Universal Robots PolyScope program: sand2.urp

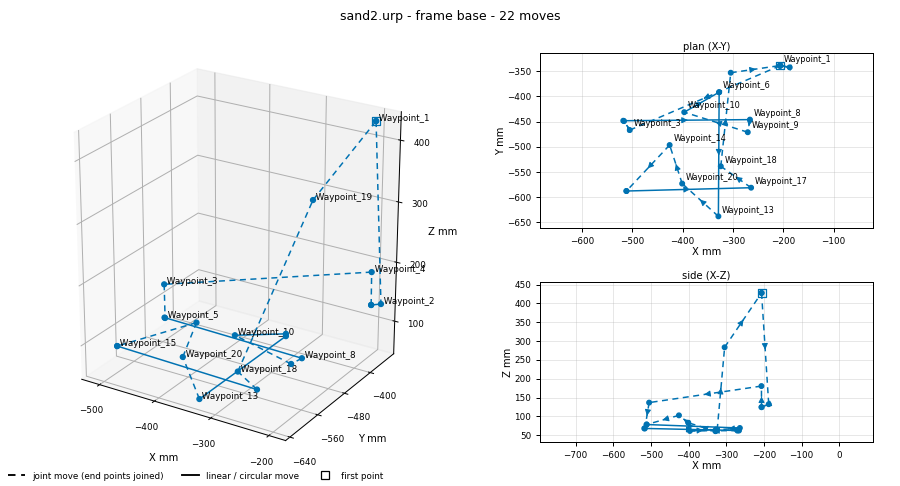
[picture p0: tool path of sand2.urp in frame base, 22 of 22 moves have a stored position in this frame; points joined in program order, loops and branches not executed]
Program sand2 (installation=default directory=/programs/archive createdIn=5.11.5.1010327 lastSavedIn=5.11.5.1010327 robotSerialNumber=20215500677)
Calibrated DH parameters: a=[0.000204, -0.239222, -0.391845, -0.000001, 0.000022, 0]; d=[0.162722, -355.808559, 353.37206, 2.570385, 0.099741, 0.099629]; alpha=[1.571124, 0.000988, 0.008295, 1.568963, -1.570303, 0]; deltaTheta=[0, -0.973091, 7.204745, 0.05153, 0, 0]
Robot Program (runOnlyOnce=false)
  MoveJ speed 60 deg/s, acceleration 80 deg/s^2 (useActiveTCP=true) feature=Base
    Waypoint Waypoint_1: TCP in base x=-206.269 y=-338.618 z=428.007 mm, rx=-2.8182 ry=-1.388 rz=0 rad; joints [-101.561, -74.063, -112.511, -83.459, 90.481, 115.929] deg
    Popup Message (haltProgram=false message=Load the cube inputType=Text)
    Waypoint Waypoint_2: TCP in base x=-187.281 y=-342.265 z=132.578 mm, rx=-2.8182 ry=-1.3882 rz=-0.0001 rad; joints [-98.674, -101.388, -141.016, -27.626, 90.232, 119.185] deg
  MoveL speed 100 mm/s, acceleration 600 mm/s^2 (useActiveTCP=true) feature=Base
    Waypoint Waypoint_7: TCP in base x=-206.272 y=-338.621 z=124.68 mm, rx=-2.8183 ry=-1.388 rz=0 rad; joints [-101.67, -103.53, -140.312, -26.186, 90.22, 116.201] deg
    URCap Finishing Tool Control (Robotiq_Copilot, Robotiq Inc.) dataModel(ToolOutputNameKey=digital_out[0], HackTriggeringContributionIsDefinedMethodKey=true)
    URCap Zero FT Sensor (Robotiq_Copilot, Robotiq Inc.) dataModel(NodeInitializedKey=true, WaitForSteadyWrenchOptionKey=false)
    URCap Find Surface (Robotiq_Copilot, Robotiq Inc.) dataModel(NodeInitializedKey=true, ZeroSensorBeforeKey=true, ls_force=10.0, ls_distance=100.0, ls_speed=5.0, ls_if_distance=false, ls_if_force=false, WaitForSteadyWrenchOptionKey=true); state(isChildrenLocked=true)
      'Add Stop conditions from the Find Surface node'
    Force Simple feature=Joint_6_name; selection=[0, 0, 1, 0, 0, 0]; wrench=[0, 0, 3, 0, 0, 0]; limitsForce=[0.15, 0.15, 0.15, 1.047198, 1.047198, 1.047198]; limitsMotion=[0.1, 0.1, 0.1, 0.349066, 0.349066, 0.349066]
      URCap Path Generator (Robotiq_Copilot, Robotiq Inc.) dataModel(pathOptionsTypeKey=TOOL_ON_ROBOT, coverageModeKey=PERIMETER_ONLY, relativePathKey=true, selectedFeatureNameKey=Actual pose, offsetTypeKey=Actual pose, PathTypeKey=FOUR_POINTS_VERTICAL, WaypointPoseKey1=[-0.20629660419563384, -0.3386300161325113, 0.12467794719703908, -2.8183538684059672, -1.3879313624712748, 7.933958590910351E-5], WaypointJointPositionsKey1=[-1.774516623062409, -1.8069839115661104, -2.4488972349192424, -0.45702049851803395, 1.5746060018745398, 2.028078014086811], WaypointPoseKey3=[-0.21004244357085544, -0.6855155317004626, 0.11340652779835002, 2.8181701273709097, 1.3883207082344338, -1.963602976327567E-4], WaypointJointPositionsKey3=[-1.6808014341985542, -2.3592393235059745, -1.4739016889725134, -0.8796152951918419, 1.5775116439677972, 2.1200337468062562], WaypointPoseKey4=[-0.5667053703425011, -0.6982977977050183, 0.1203185558229202, 2.818031624647423, 1.3883496686721377, -2.3680285315842763E-4], WaypointJointPositionsKey4=[-2.1036509005491766, -2.8258939963203815, -0.5103127280502875, -1.3765599820875805, 1.5793118514988338, 1.6940088214635205], WaypointPoseKey2=[-0.5685400620358461, -0.32892856911544577, 0.1182503073618568, 2.818063926809957, 1.3885574833411425, -2.2199273126068995E-4], WaypointJointPositionsKey2=[-2.412473690950604, -2.2446352860444456, -1.6836503159348153, -0.7843915989155441, 1.5769781191650418, 1.388733307698494], urcapVersion=1.22.1); state(isChildrenLocked=true)
        URCap Point (Robotiq_Copilot, Robotiq Inc.) dataModel(pose=[-0.20629660419563384, -0.3386300161325113, 0.12467794719703908, -2.8183538684059672, -1.3879313624712748, 7.933958590910351E-5], joint_positions=[-1.774516623062409, -1.8069839115661104, -2.4488972349192424, -0.45702049851803395, 1.5746060018745398, 2.028078014086811])
        URCap Point (Robotiq_Copilot, Robotiq Inc.) dataModel(pose=[-0.5685400620358461, -0.32892856911544577, 0.1182503073618568, 2.818063926809957, 1.3885574833411425, -2.2199273126068995E-4], joint_positions=[-2.412473690950604, -2.2446352860444456, -1.6836503159348153, -0.7843915989155441, 1.5769781191650418, 1.388733307698494])
        URCap Point (Robotiq_Copilot, Robotiq Inc.) dataModel(pose=[-0.21004244357085544, -0.6855155317004626, 0.11340652779835002, 2.8181701273709097, 1.3883207082344338, -1.963602976327567E-4], joint_positions=[-1.6808014341985542, -2.3592393235059745, -1.4739016889725134, -0.8796152951918419, 1.5775116439677972, 2.1200337468062562])
        URCap Point (Robotiq_Copilot, Robotiq Inc.) dataModel(pose=[-0.5667053703425011, -0.6982977977050183, 0.1203185558229202, 2.818031624647423, 1.3883496686721377, -2.3680285315842763E-4], joint_positions=[-2.1036509005491766, -2.8258939963203815, -0.5103127280502875, -1.3765599820875805, 1.5793118514988338, 1.6940088214635205])
  MoveJ speed 60 deg/s, acceleration 80 deg/s^2 (useActiveTCP=true) feature=Base
    Waypoint Waypoint_7: TCP in base x=-206.272 y=-338.621 z=124.68 mm, rx=-2.8183 ry=-1.388 rz=0 rad; joints [-101.67, -103.53, -140.312, -26.186, 90.22, 116.201] deg
    Waypoint Waypoint_4: TCP in base x=-206.628 y=-339.081 z=180.69 mm, rx=-2.8185 ry=-1.3836 rz=-0.0007 rad; joints [-101.68, -93.905, -137.581, -38.641, 90.262, 116.28] deg
  MoveJ speed 60 deg/s, acceleration 80 deg/s^2 (useActiveTCP=true) feature=Base
    Waypoint Waypoint_3: TCP in base x=-504.833 y=-466.759 z=136.802 mm, rx=-1.4822 ry=0.6139 rz=0.614 rad; joints [-121.492, -151.792, -47.283, -160.609, 58.713, 224.343] deg
    Waypoint Waypoint_5: TCP in base x=-516.197 y=-448.962 z=68.19 mm, rx=-1.4821 ry=0.6139 rz=0.6139 rad; joints [-122.967, -155.557, -50.4, -153.726, 57.296, 224.364] deg
  URCap Find Surface (Robotiq_Copilot, Robotiq Inc.) dataModel(NodeInitializedKey=true, ZeroSensorBeforeKey=true, ls_force=10.0, ls_distance=100.0, ls_speed=5.0, WaitForSteadyWrenchOptionKey=true, ls_if_distance=false, ls_if_force=false); state(isChildrenLocked=true)
    'Add Stop conditions from the Find Surface node'
  Force Simple feature=Joint_6_name; selection=[0, 0, 1, 0, 0, 0]; wrench=[0, 0, 1, 0, 0, 0]; limitsForce=[0.15, 0.15, 0.15, 1.047198, 1.047198, 1.047198]; limitsMotion=[0.1, 0.1, 0.1, 0.349066, 0.349066, 0.349066]
    MoveL speed 60 mm/s, acceleration 600 mm/s^2 (useActiveTCP=true) feature=Base
      Waypoint Waypoint_11: TCP in base x=-517.708 y=-448.208 z=68.219 mm, rx=-1.4821 ry=0.614 rz=0.6139 rad; joints [-123.097, -155.632, -50.239, -153.808, 57.165, 224.365] deg
      Waypoint Waypoint_8: TCP in base x=-266.257 y=-446.005 z=62.63 mm, rx=-1.4821 ry=0.6144 rz=0.6139 rad; joints [-103.202, -138.545, -87.527, -133.849, 77.187, 224.556] deg
  MoveJ speed 60 deg/s, acceleration 80 deg/s^2 (useActiveTCP=true) feature=Base
    Waypoint Waypoint_9: TCP in base x=-270.568 y=-471.038 z=62.458 mm, rx=-1.4822 ry=0.6139 rz=0.6139 rad; joints [-103.059, -140.977, -82.312, -136.634, 77.304, 224.524] deg
    Waypoint Waypoint_10: TCP in base x=-396.671 y=-431.249 z=61.533 mm, rx=-1.6291 ry=0.8608 rz=-1.5805 rad; joints [-127.01, -143.859, -76.086, -139.656, 141.376, 147.667] deg
  MoveL speed 250 mm/s, acceleration 1200 mm/s^2 (useActiveTCP=true) feature=Base
    Waypoint Waypoint_6: TCP in base x=-327.39 y=-391.56 z=65.51 mm, rx=-1.629 ry=0.8608 rz=-1.5805 rad; joints [-123.845, -135.688, -92.857, -130.988, 144.58, 147.788] deg
    URCap Find Surface (Robotiq_Copilot, Robotiq Inc.) dataModel(NodeInitializedKey=true, ZeroSensorBeforeKey=true, ls_force=10.0, ls_distance=100.0, ls_speed=5.0, WaitForSteadyWrenchOptionKey=true, ls_if_distance=false, ls_if_force=false); state(isChildrenLocked=true)
      'Add Stop conditions from the Find Surface node'
    Force Simple feature=Joint_6_name; selection=[0, 0, 1, 0, 0, 0]; wrench=[0, 0, 1, 0, 0, 0]; limitsForce=[0.15, 0.15, 0.15, 1.047198, 1.047198, 1.047198]; limitsMotion=[0.1, 0.1, 0.1, 0.349066, 0.349066, 0.349066]
      MoveL speed 60 mm/s, acceleration 600 mm/s^2 (useActiveTCP=true) feature=Base
        Waypoint Waypoint_12: TCP in base x=-327.379 y=-391.583 z=61.531 mm, rx=-1.6292 ry=0.8608 rz=-1.5805 rad; joints [-123.844, -136.089, -92.862, -130.571, 144.584, 147.793] deg
        Waypoint Waypoint_13: TCP in base x=-328.883 y=-638.051 z=60.857 mm, rx=-2.0082 ry=0.3792 rz=-1.9571 rad; joints [-113.687, -158.85, -44.386, -155.599, 154.435, 114.309] deg
    MoveJ speed 60 deg/s, acceleration 80 deg/s^2 (useActiveTCP=true) feature=Base
      Waypoint Waypoint_20: TCP in base x=-400.771 y=-573.011 z=83.242 mm, rx=-1.958 ry=0.4443 rz=-1.9994 rad; joints [-120.966, -156.796, -45.744, -160.68, 149.608, 112.129] deg
      Waypoint Waypoint_14: TCP in base x=-425.676 y=-496.485 z=102.964 mm, rx=1.1538 ry=-1.3748 rz=1.4281 rad; joints [-124.203, -132.766, -90.964, -137.131, 232.086, 103.899] deg
      Waypoint Waypoint_15: TCP in base x=-511.481 y=-587.765 z=78.601 mm, rx=1.1164 ry=-1.3919 rz=1.3957 rad; joints [-125.535, -148.505, -63.116, -149.198, 233.273, 103.952] deg
    URCap Find Surface (Robotiq_Copilot, Robotiq Inc.) dataModel(NodeInitializedKey=true, ZeroSensorBeforeKey=true, ls_force=10.0, ls_distance=100.0, ls_speed=5.0, WaitForSteadyWrenchOptionKey=true, ls_if_distance=false, ls_if_force=false); state(isChildrenLocked=true)
      'Add Stop conditions from the Find Surface node'
    Force Simple feature=Joint_6_name; selection=[0, 0, 1, 0, 0, 0]; wrench=[0, 0, 1, 0, 0, 0]; limitsForce=[0.15, 0.15, 0.15, 1.047198, 1.047198, 1.047198]; limitsMotion=[0.1, 0.1, 0.1, 0.349066, 0.349066, 0.349066]
      MoveL speed 60 mm/s, acceleration 600 mm/s^2 (useActiveTCP=true) feature=Base
        Waypoint Waypoint_16: TCP in base x=-511.48 y=-587.758 z=78.584 mm, rx=1.1165 ry=-1.3919 rz=1.3957 rad; joints [-125.535, -148.506, -63.117, -149.196, 233.271, 103.952] deg
        Waypoint Waypoint_17: TCP in base x=-263.924 y=-581.188 z=69.357 mm, rx=1.1165 ry=-1.3919 rz=1.3958 rad; joints [-104.804, -132.622, -98.496, -129.775, 254.098, 104.182] deg
    URCap Finishing Tool Control (Robotiq_Copilot, Robotiq Inc.) dataModel(FinishingToolStateKey=false, ToolOutputNameKey=digital_out[0], HackTriggeringContributionIsDefinedMethodKey=true)
    MoveJ speed 60 deg/s, acceleration 80 deg/s^2 (useActiveTCP=true) feature=Base
      Waypoint Waypoint_18: TCP in base x=-324.128 y=-538.628 z=64.354 mm, rx=1.1164 ry=-1.3918 rz=1.3957 rad; joints [-112.416, -132.876, -99.115, -128.885, 246.496, 104.047] deg
      Waypoint Waypoint_19: TCP in base x=-304.37 y=-352.926 z=283.741 mm, rx=-2.1974 ry=2.152 rz=0.0807 rad; joints [-113.684, -117.514, -87.457, -249.545, 271.021, 65.463] deg
  MoveJ speed 60 deg/s, acceleration 80 deg/s^2 (useActiveTCP=true) feature=Base
    Waypoint Waypoint_1: TCP in base x=-206.269 y=-338.618 z=428.007 mm, rx=-2.8182 ry=-1.388 rz=0 rad; joints [-101.561, -74.063, -112.511, -83.459, 90.481, 115.929] deg
  SuppressedNode
    MoveJ speed 60 deg/s, acceleration 80 deg/s^2 (useActiveTCP=true) feature=Base
      Waypoint Waypoint_4: TCP in base x=-525.053 y=-216.53 z=116.815 mm, rx=-1.5142 ry=0.9781 rz=-1.5142 rad; joints [-149.128, -139.618, -74.936, -145.787, 121.181, 155.098] deg
  SuppressedNode
    URCap Multipoint Path (Robotiq_Copilot, Robotiq Inc.) dataModel(NodeInitializedKey=true, pathOptionsTypeKey=TOOL_ON_ROBOT, waypointIndexKey=4, SPEED_VALUE=60, HackTriggeringContributionIsDefinedMethodKey=true, urcapVersion=1.22.1)
      URCap Waypoint (Robotiq_Copilot, Robotiq Inc.) dataModel(NodeIndexKey=1, RenamedTitleKey=UnrenamedTitle, pose=[-0.46978261103261726, -0.16844710267869106, 0.1168867034882474, -1.5586921977868937, 0.9328885874148277, -1.5509326951155455], jointPositions=[-2.6239750749989774, -2.307789293024514, -1.5640154177641614, -2.4161803968612894, 2.0867638040135716, 2.6474263722654925], waypointType=CURVE, waypointIndex=0, initialized=true, urcapVersion=1.22.1)
      URCap Waypoint (Robotiq_Copilot, Robotiq Inc.) dataModel(pose=[-0.4587585249204176, -0.43646083988176626, 0.1169249537563768, -1.785675246785113, 0.6795322510770658, -1.7706886463906304], jointPositions=[-2.2850269277871242, -2.5454670750737414, -1.0893249131228568, -2.6593833558941355, 2.4112405226427716, 2.304287772798501], waypointType=LINE, waypointIndex=0, initialized=true, NodeIndexKey=2, RenamedTitleKey=UnrenamedTitle, urcapVersion=1.22.1)
      URCap Waypoint (Robotiq_Copilot, Robotiq Inc.) dataModel(NodeIndexKey=3, RenamedTitleKey=UnrenamedTitle, pose=[-0.5244673627388496, -0.2742524201709816, 0.11689590126719628, -1.7855589020629918, 0.679551965066376, -1.7706531031839516], jointPositions=[-2.5261688322632736, -2.481941308010927, -1.2171111467983238, -2.590743410546766, 2.170498860232936, 2.3074613956460106], waypointType=LINE, waypointIndex=0, initialized=true, urcapVersion=1.22.1)
  SuppressedNode
    MoveJ speed 60 deg/s, acceleration 80 deg/s^2 (useActiveTCP=true) feature=Base
      Waypoint Waypoint_5: TCP in base x=-668.757 y=-381.561 z=120.836 mm, rx=1.1942 ry=-1.2322 rz=1.2322 rad; joints [-146.452, -147.427, -58.584, -153.108, 213.802, 92.834] deg
  SuppressedNode
    URCap Multipoint Path (Robotiq_Copilot, Robotiq Inc.) dataModel(NodeInitializedKey=true, pathOptionsTypeKey=TOOL_ON_ROBOT, SPEED_VALUE=60, waypointIndexKey=3, HackTriggeringContributionIsDefinedMethodKey=true, urcapVersion=1.22.1)
      URCap Waypoint (Robotiq_Copilot, Robotiq Inc.) dataModel(pose=[-0.6687417922557757, -0.38156646353184936, 0.1207900175721562, 1.194242294591316, -1.232318957369504, 1.2323037155227854], jointPositions=[-2.5560443392566894, -2.5730936628743724, -1.0225160828281936, -2.6722180449841155, 3.7315478772490542, 1.6202727383200735], waypointType=CURVE, waypointIndex=0, initialized=true, NodeIndexKey=1, RenamedTitleKey=UnrenamedTitle, urcapVersion=1.22.1)
      URCap Waypoint (Robotiq_Copilot, Robotiq Inc.) dataModel(pose=[-0.40381107400266475, -0.3815787704989514, 0.12078674530058967, 1.1942586617152338, -1.2322856393078285, 1.2322932044982344], jointPositions=[-2.255100698114216, -2.1261101664285773, -1.9024833295513712, -2.248045227522269, 4.03471213212066, 1.6120633716471122], waypointType=LINE, waypointIndex=0, initialized=true, NodeIndexKey=2, RenamedTitleKey=UnrenamedTitle, urcapVersion=1.22.1)
      URCap Waypoint (Robotiq_Copilot, Robotiq Inc.) dataModel(NodeIndexKey=3, RenamedTitleKey=UnrenamedTitle, pose=[-0.5267445821917994, -0.3353892075077195, 0.12080665354845467, 1.194246265841587, -1.2322959935554332, 1.2322953440029232], jointPositions=[-2.4852409944789606, -2.268679223280569, -1.6274892138186559, -2.3757156340447563, 3.804019056086524, 1.6161677359875088], waypointType=LINE, waypointIndex=0, initialized=true, urcapVersion=1.22.1)
  SuppressedNode
    MoveL speed 250 mm/s, acceleration 1200 mm/s^2 (useActiveTCP=true) feature=Base
      Waypoint Waypoint_6: TCP in base x=-548.582 y=-380.65 z=223.769 mm, rx=-3.0572 ry=-0.723 rz=0.0001 rad; joints [-133.698, -120.992, -90.454, -58.581, 90.428, 109.851] deg
